PROGRAM PRG_TEST
VAR
    _testSuite : TcUnitContext;
END_VAR

_testSuite.Run();
_testSuite.RtcSynchronize(true, '', 60);

END_PROGRAM

(* stored: Version 1.1.0.1, ProductVersion 3.1.4024.12
   POU PRG_TEST: Id {2dc1ad44-fabf-06dc-3389-3a5eaed67bf6}, SpecialFunc None *)
